FUNCTION_BLOCK _HRESULT_TestSuite EXTENDS TcUnit.FB_TestSuite
VAR
END_VAR

TestAddress();
TestClearReference();
TestClone();
TestTypeNameReturnsExpected();
TestIdentifierReturnsExpected();
TestMakeReferenceToFollowsReference();
TestMakeReferenceToUpdatesReference();
TestSize();
TestValueReturnsExpectedAfterInit();
TestValueReturnsExpectedAfterChange();
TestSerializeTypeWith();
TestSerializeWith();
TestTryDeserializeFrom();
TestTryMakeReferenceToFollowsReference();
TestTryMakeReferenceToUpdatesReference();

METHOD PUBLIC TestAddress
VAR
    _type : _HRESULT(S_OK);
    notExpected : PVOID := 0;
    actual : PVOID;
END_VAR
TEST('TestAddress');

actual := _type.Address;

AssertFalse(
    Condition := (notExpected = actual),
    Message := 'Type did not return a valid address.'
);

TEST_FINISHED();
END_METHOD

METHOD PUBLIC TestClearReference
VAR
    _type : _HRESULT(S_OK);
	target : HRESULT := S_OK;
    expected : HRESULT := S_OK;
    actual : HRESULT;
END_VAR
TEST('TestClearReference');

_type.MakeReferenceTo(target);
_type.ClearReference();
target := S_FALSE;

actual := _type.Value;

AssertEquals(
    Expected := expected,
    Actual := actual,
    Message := 'Value did not follow target change'
);

TEST_FINISHED();
END_METHOD

METHOD PUBLIC TestClone
VAR
    _type : _HRESULT(S_OK);
	clone : I_Datatype;
	isValidClone : BOOL;
	compareResult : DINT;
END_VAR
TEST('TestClone');

clone := _type.Clone();

isValidClone := clone <> 0;

IF isValidClone THEN
	compareResult := memcmp(_type.Address, clone.Address, clone.Size);
END_IF

AssertTrue(
	Condition := isValidClone,
	Message := 'Clone did not produce a clone'
);

AssertEquals_DINT(
	Expected := 0,
    Actual := compareResult,
    Message := 'Clone did not return a valid clone.'
);

clone.Dispose();

TEST_FINISHED();
END_METHOD

METHOD PUBLIC TestIdentifierReturnsExpected
VAR
    _type : _HRESULT(S_OK);
    expected : STRING := 'HRESULT';
    actual : STRING;
END_VAR
TEST('TestIdentifierReturnsExpected');

actual := _type.Identifier;

AssertEquals_STRING(
    Expected := expected,
    Actual := actual,
    Message := 'Type did not return correct iec type.'
);

TEST_FINISHED();
END_METHOD

METHOD PUBLIC TestMakeReferenceToFollowsReference
VAR
    _type : _HRESULT(S_OK);
	target : HRESULT := S_OK;
    expected : HRESULT := S_FALSE;
    actual : HRESULT;
END_VAR
TEST('TestMakeReferenceToFollowsReference');

_type.MakeReferenceTo(target);
target := S_FALSE;

actual := _type.Value;

AssertEquals(
    Expected := expected,
    Actual := actual,
    Message := 'Value did not follow target change'
);

TEST_FINISHED();
END_METHOD

METHOD PUBLIC TestMakeReferenceToUpdatesReference
VAR
    _type : _HRESULT(S_OK);
	target : HRESULT := S_OK;
    expected : HRESULT := S_FALSE;
    actual : HRESULT;
END_VAR
TEST('TestMakeReferenceToUpdatesReference');

_type.MakeReferenceTo(target);
_type.Value := S_FALSE;

actual := target;

AssertEquals(
    Expected := expected,
    Actual := actual,
    Message := 'Value did not update target'
);

TEST_FINISHED();
END_METHOD

METHOD PUBLIC TestSerializeTypeWith
VAR
    _type : _HRESULT(S_OK);
    serializer : JsonSerializer;
    expected : STRING(500) := '{"typeName":"ALIAS","identifier":"HRESULT","baseDatatype":{"typeName":"DINT","minValue":-2147483648,"maxValue":2147483647,"isSigned":true,"isFloat":false}}';
    actual : STRING(500);
END_VAR
TEST('TestSerializeTypeWith');

serializer.Reset();
_type.SerializeTypeWith(serializer);
serializer.TryGetSerializedData(ADR(actual), SIZEOF(actual));

AssertEquals_STRING(
    Expected := expected,
    Actual := actual,
    Message := 'Serialization of type did not return correct string.'
);

TEST_FINISHED();
END_METHOD

METHOD PUBLIC TestSerializeWith
VAR
    _type : _HRESULT(S_FALSE);
    serializer : JsonSerializer;
    expected : STRING := '1';
    actual : STRING(500);
END_VAR
TEST('TestSerializeWith');

serializer.Reset();
_type.SerializeWith(serializer);
serializer.TryGetSerializedData(ADR(actual), SIZEOF(actual));

AssertEquals_STRING(
    Expected := expected,
    Actual := actual,
    Message := 'Serialization of type data did not return correct string.'
);

TEST_FINISHED();
END_METHOD

METHOD PUBLIC TestSize
VAR
    _type : _HRESULT(S_OK);
    expected : UDINT := SIZEOF(HRESULT);
    actual : UDINT;
END_VAR
TEST('TestSize');

actual := _type.Size;

AssertEquals_UDINT(
    Expected := Expected,
    Actual := actual,
    Message := 'Type did not return the correct size.'
);

TEST_FINISHED();
END_METHOD

METHOD PUBLIC TestTryDeserializeFrom
VAR
    deserializer : JsonDeserializer;
    feedback : DeserializerFeedback;
    json : STRING := '0';
    _type : _HRESULT(S_OK);
    expected : HRESULT := S_OK;
    actual : HRESULT;
 END_VAR
TEST('TestTryDeserializeFrom');

deserializer.Reset();
deserializer.TryLoad(json);
_type.TryDeserializeFrom(Deserializer, Feedback);

actual := _type.Value;

AssertEquals(
    Expected := expected,
    Actual := actual,
    Message := 'Type did not deserialize correctly.'
);

TEST_FINISHED();
END_METHOD

METHOD PUBLIC TestTryMakeReferenceToFollowsReference
VAR
    _type : _HRESULT(S_OK);
	target : _HRESULT(S_OK);
    expected : HRESULT := S_FALSE;
    actual : HRESULT;
END_VAR
TEST('TestTryMakeReferenceToFollowsReference');

_type.TryMakeReferenceTo(target);
target.Value := S_FALSE;

actual := _type.Value;

AssertEquals(
    Expected := expected,
    Actual := actual,
    Message := 'Value did not follow target change'
);

TEST_FINISHED();
END_METHOD

METHOD PUBLIC TestTryMakeReferenceToUpdatesReference
VAR
    _type : _HRESULT(S_OK);
	target : _HRESULT(S_OK);
    expected : HRESULT := S_FALSE;
    actual : HRESULT;
END_VAR
TEST('TestTryMakeReferenceToUpdatesReference');

_type.TryMakeReferenceTo(target);
_type.Value := S_FALSE;

actual := target.Value;

AssertEquals(
    Expected := expected,
    Actual := actual,
    Message := 'Value did not update target'
);

TEST_FINISHED();
END_METHOD

METHOD PUBLIC TestTypeNameReturnsExpected
VAR
    _type : _HRESULT(S_OK);
    expected : STRING := 'ALIAS';
    actual : STRING;
END_VAR
TEST('TestTypeNameReturnsExpected');

actual := _type.TypeName;

AssertEquals_STRING(
    Expected := expected,
    Actual := actual,
    Message := 'Type did not return correct iec type.'
);

TEST_FINISHED();
END_METHOD

METHOD PUBLIC TestValueReturnsExpectedAfterChange
VAR
    _type : _HRESULT(S_OK);
    expected : HRESULT := S_FALSE;
    actual : HRESULT;
END_VAR
TEST('TestValueReturnsExpectedAfterChange');

_type.Value := S_FALSE;

actual := _type.Value;

AssertEquals(
    Expected := expected,
    Actual := actual,
    Message := 'Expected value not returned after change.'
);

TEST_FINISHED();
END_METHOD

METHOD PUBLIC TestValueReturnsExpectedAfterInit
VAR
    _type : _HRESULT(S_FALSE);
    expected : HRESULT := S_FALSE;
    actual : HRESULT;
END_VAR
TEST('TestValueReturnsExpectedAfterInit');

actual := _type.Value;

AssertEquals(
    Expected := expected,
    Actual := actual,
    Message := 'Expected value not returned after Init.'
);

TEST_FINISHED();
END_METHOD

END_FUNCTION_BLOCK

(* stored: Version 1.1.0.1, ProductVersion 3.1.4024.12
   POU _HRESULT_TestSuite: Id {6bfd07a7-b13c-494a-8264-4ea3d1a239ba}, SpecialFunc None
   Method TestAddress: Id {a886895d-bfd1-466a-98cf-238e5d115f24}
   Method TestClearReference: Id {57199a35-db2d-491d-ab9b-5eee170d3b12}
   Method TestClone: Id {d5ee2fae-ee6a-4b51-a259-9279a1276c0d}
   Method TestIdentifierReturnsExpected: Id {6bbec32f-e889-44c0-8a7b-68f185b6e073}
   Method TestMakeReferenceToFollowsReference: Id {fdb15262-43c4-47bb-913d-d36ff376f7b8}
   Method TestMakeReferenceToUpdatesReference: Id {9cc402b6-155f-421b-8e66-15930d2a6662}
   Method TestSerializeTypeWith: Id {7fdb9c86-c305-4171-b273-878d60e9ee38}
   Method TestSerializeWith: Id {4ab0cca4-ac2b-4a83-bc9f-075252bc5ccf}
   Method TestSize: Id {1481a4dc-3543-4470-946e-cf10eefc4c7e}
   Method TestTryDeserializeFrom: Id {2e55a048-0c4c-4cef-927f-6225b2709caa}
   Method TestTryMakeReferenceToFollowsReference: Id {b67ad62e-274c-44c0-bec0-2aa9fb396ad7}
   Method TestTryMakeReferenceToUpdatesReference: Id {0139f5b5-f23e-4705-8073-edadb8149b8e}
   Method TestTypeNameReturnsExpected: Id {bebb11dd-166d-4275-8227-9b94cd0ad2ce}
   Method TestValueReturnsExpectedAfterChange: Id {0f424c01-5e11-4a42-9a54-0dd777a8d801}
   Method TestValueReturnsExpectedAfterInit: Id {dc31a871-6c0d-4440-9662-da6b5a366d66} *)
